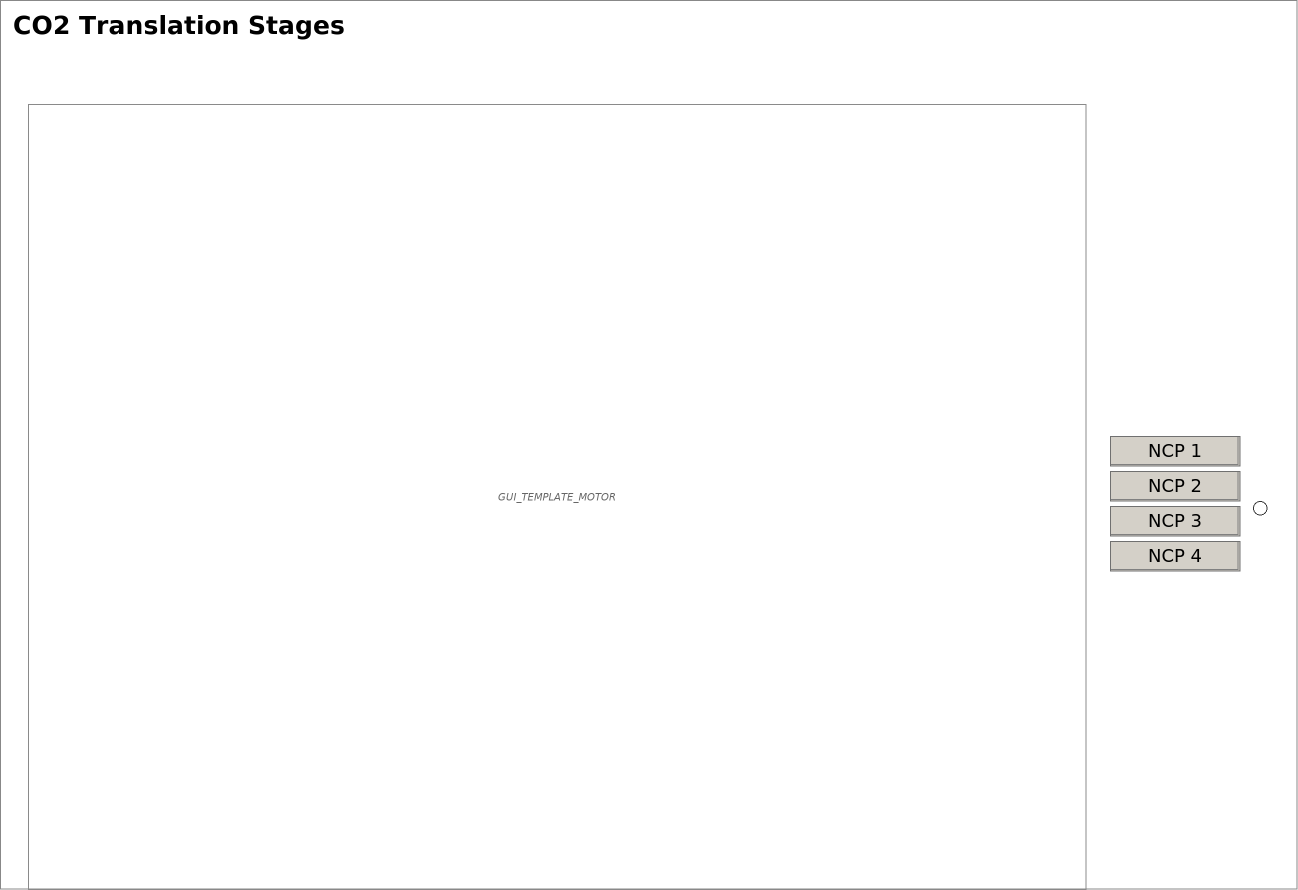
VISUALIZATION VISU_HMI_CO2_TRANS_STAGES  // 1298x890
    Label (10,10 379x30), "CO2 Translation Stages"
    Frame (28,104 1058x786)
        shows GUI_TEMPLATE_MOTOR(m_Instance := MAIN.nott_ics.CO2TransStages.ptrNCPs[MAIN.nott_ics.CO2TransStages.guiNCPsIndex]^)
    RadioButton (1251,438 47x140), variable: MAIN.nott_ics.CO2TransStages.guiNCPsIndex-1
        Areas[0]: Text=Radiobutton
        Areas[1]: Text=Radiobutton
    Button (1110,436 130x30), "NCP 1"
        OnMouseClick: execute { MAIN.nott_ics.CO2TransStages.guiNCPsIndex := 1; }
    Button (1110,471 130x30), "NCP 2"
        OnMouseClick: execute { MAIN.nott_ics.CO2TransStages.guiNCPsIndex := 2; }
    Button (1110,506 130x30), "NCP 3"
        OnMouseClick: execute { MAIN.nott_ics.CO2TransStages.guiNCPsIndex := 3; }
    Button (1110,541 130x30), "NCP 4"
        OnMouseClick: execute { MAIN.nott_ics.CO2TransStages.guiNCPsIndex := 4; }
END_VISUALIZATION

(* stored: Version 1.1.0.1, ProductVersion 3.1.4024.14
   Visu VISU_HMI_CO2_TRANS_STAGES: Id {889b7fff-6a8c-4816-b539-43a1f29dee23} *)
